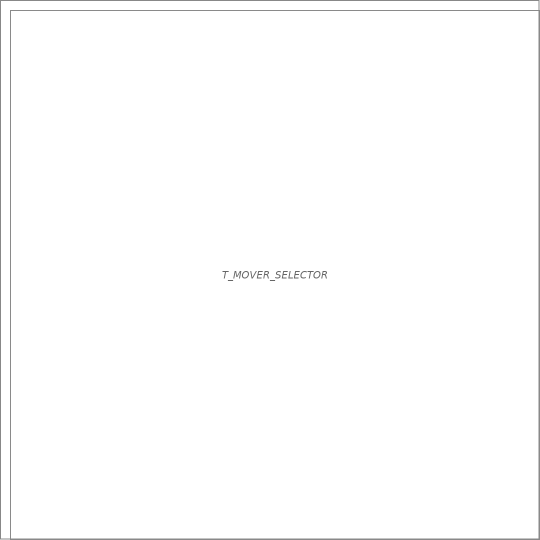
VISUALIZATION SELECTOR_VISU  // 540x540
    Frame (10,10 530x530)
        shows T_MOVER_SELECTOR(Control := GVL_XTS.SelectorCtrl, State := GVL_XTS.SelectorState, sState := MAIN.sSelectorState, sResult := MAIN.sSelectorResult)
END_VISUALIZATION

(* stored: Version 1.1.0.1
   Visu SELECTOR_VISU: Id {19b65231-913d-486e-b869-9fd1d1a713b8} *)
